// TIA Portal V20 export
TYPE "typeEmInterlock"
// stored: Access Published, Namespace Unit1
   STRUCT
      General { ExternalAccessible := 'False'; ExternalVisible := 'False'; ExternalWritable := 'False'} : "Unit1.typeEmInterlockParameters";
      EM0 { ExternalAccessible := 'False'; ExternalVisible := 'False'; ExternalWritable := 'False'} : "Unit1.typeEmInterlockParameters";
      EM1 { ExternalAccessible := 'False'; ExternalVisible := 'False'; ExternalWritable := 'False'} : "Unit1.typeEmInterlockParameters";
      EM2 { ExternalAccessible := 'False'; ExternalVisible := 'False'; ExternalWritable := 'False'} : "Unit1.typeEmInterlockParameters";
      EM3 { ExternalAccessible := 'False'; ExternalVisible := 'False'; ExternalWritable := 'False'} : "Unit1.typeEmInterlockParameters";
      EM4 { ExternalAccessible := 'False'; ExternalVisible := 'False'; ExternalWritable := 'False'} : "Unit1.typeEmInterlockParameters";
      EM5 { ExternalAccessible := 'False'; ExternalVisible := 'False'; ExternalWritable := 'False'} : "Unit1.typeEmInterlockParameters";
      EM6 { ExternalAccessible := 'False'; ExternalVisible := 'False'; ExternalWritable := 'False'} : "Unit1.typeEmInterlockParameters";
      EM7 { ExternalAccessible := 'False'; ExternalVisible := 'False'; ExternalWritable := 'False'} : "Unit1.typeEmInterlockParameters";
   END_STRUCT;
   // // General.Lreal[0] : CPM
   // // General.Lreal[1] : Electrode Width
   // // General.Lreal[2] : Tab Width
   // // General.Lreal[3] : Electrode ~ TabWidth
   // // General.Lreal[4] : Anode Gap Width
   // // General.Lreal[5] : Cathode Gap Width
   // // General.Lreal[6] : Anode Thinkness
   // // General.Lreal[7] : Cathode Thinkness
   // // General.Lreal[8] : Separator Thinkness
   // // General.Lreal[9] : Jelly Roll Width
   // // EM0.Lreal[0] : SepaUnwinderRadious
   // // EM1.Lreal[0] : SepaUnwinderRadious
   // // EM2."Bool"[3] : DancerPneumaticRegulatorReduceRequst
   // // EM2."Bool"[4] : TopUnwinderRewindingRequset
   // // EM2."Bool"[5] : BottomUnwinderRewindingRequset
   // // EM3."Bool"[3] : DancerPneumaticRegulatorReduceDone
   // // EM3.Lreal[0] : TargetDancerAngle
   // // EM3.Lreal[1] : CurrentDancerAngle
   // // EM3.Lreal[2] : DancerLenth
   // // EM3.Lreal[3] : Compasator Storke
   // // EM6."Bool"[3] : JellyRollStackTableOut
END_TYPE
